// TIA Portal V20 export
VAR_GLOBAL   // PLC tag table "LGR_Const_AlarmClass"
END_VAR
VAR_GLOBAL CONSTANT   // user constants
   ALARM_FAULT : UInt := 1;   // Alarm Class : Fault
   ALARM_WARN : UInt := 2;   // Alarm Class : Warnning
   ALM_GROUP_HARDWARE : UInt := 10;   // Alarm Group : Hardware
   ALM_GROUP_PROC : UInt := 40;   // Alarm Group : Process
   ALM_GROUP_TIMEOUT : UInt := 50;   // Alarm Group : TimeOut
   ALM_GROUP_COMM : UInt := 70;   // Alarm Group : Communication
   ALM_GROUP_SENSOR : UInt := 80;   // Alarm Group : Sensor
   ALM_GROUP_SAFETY : UInt := 90;   // Alarm Group : Safety
   ALM_GROUP_CONFIG : UInt := 1;   // Alarm Group : Configuration
   ALM_GROUP_DRIVE : UInt := 20;   // Alarm Group : Drive
   ALM_GROUP_INIT : UInt := 30;   // Alarm Group : Initializing
   ALM_GROUP_DATA : UInt := 60;   // Alarm Group : Data
   ALARM_EVENT : UInt := 3;
   ALARM_FAULT_TRACKING : UInt := 4;   // Alarm Class : Fault (Tracking)
END_VAR
